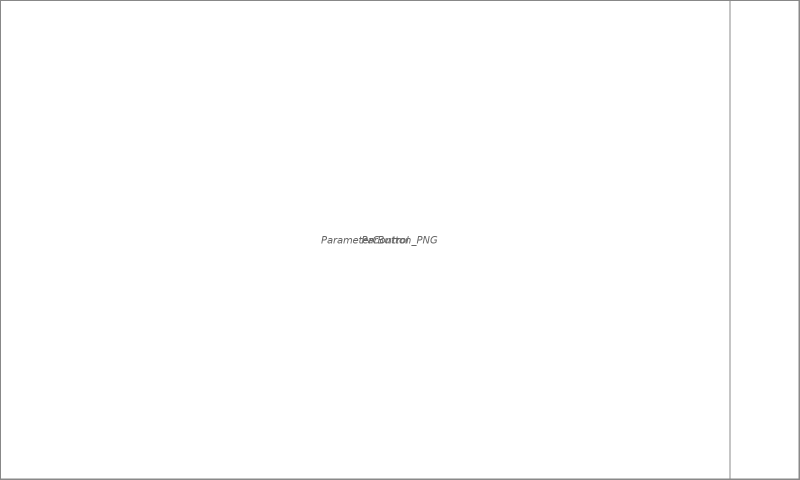
VISUALIZATION Parameter_PNG  // 800x480
VAR_IN_OUT
	bCmdParameter : BOOL ; // Return from parameter screen
END_VAR
    Frame (0,0 800x480)
        shows ParButton_PNG(bCmdParameter := bCmdParameter)
    Frame (0,0 730x480)
        shows ParameterControl()
END_VISUALIZATION

(* stored: Version 1.1.0.1, ProductVersion 3.1.4024.5
   Visu Parameter_PNG: Id {9fbd6c62-8c6c-4f75-a011-1c90743c0900} *)
